{attribute 'GeneratedUsingTerminal: EK1100-0000-0018'}
{attribute addProperty BoxType "EK1100-0000-0018"}
{attribute addProperty Id "Beckhoff_EP8xxxEK1122Beckhoff_EP8xxxEK1122_8E7F58BE250"}
{attribute addProperty CRC "863781280"}
{attribute addProperty Size "250"}
TYPE Beckhoff_EP8xxx_337C41A0 EXTENDS EK1100_1FC0878B :
STRUCT
	{attribute addProperty Name "Beckhoff_EP8xxxEK1122"}
	{attribute addProperty PreviousPort "Beckhoff EP8xxx : B"}
	Beckhoff_EP8xxxEK1122 : Beckhoff_EP8xxxEK1122_8E7F58BE;
END_STRUCT
END_TYPE

(* stored: Version 1.2.0.0, ProductVersion 3.1.4024.9
   DUT Beckhoff_EP8xxx_337C41A0: Id {c199556a-c0c3-4e1e-b22d-7c3652ba2f53} *)
